FUNCTION_BLOCK SUB_COLOR (* COLOR Subtraction *)
  (* Standard: 61131-3 *)
  (* Version 0.0, 2004-12-15, JHC, Rockwell Automation, Converted from SRC format. *)
  (* Compiler header: package fb.rt.plc.math; *)
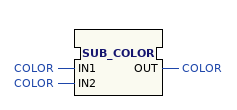
  VAR_INPUT
    IN1 : COLOR; (* Minuend *)
    IN2 : COLOR; (* Subtrahend *)
  END_VAR
  VAR_OUTPUT
    OUT : COLOR; (* Difference *)
  END_VAR
END_FUNCTION_BLOCK
